(* CODESYS project Acionamento da esteira transportadora.project

Project tree, tasks and I/O mapping:
  Device : CODESYS Control Win V3, 3S - Smart Software Solutions GmbH, order no. 305021, version 3.5.11.30
    application Application
      libraries: Standard, * (System)
      task MainTask (cyclic, interval t#20ms, priority 1) calls PLC_PRG
      program PLC_PRG [LD]
      Symbols
*)

// Device/Application/PLC_PRG
PROGRAM PLC_PRG
VAR
	Start:BOOL;
	Stop:BOOL;
	Emergencia:BOOL;
	Sensor:BOOL;
	Start_Light:BOOL;
	Stop_Light:BOOL;
	Esteira:BOOL;
	
	
END_VAR

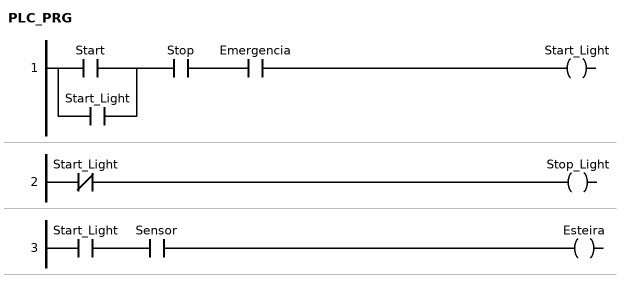
// NETWORK 1
Start_Light := (Start OR Start_Light) AND Stop AND Emergencia;

// NETWORK 2
Stop_Light := NOT Start_Light;

// NETWORK 3
Esteira := Start_Light AND Sensor;

END_PROGRAM
